(* Logix 5000 project; controller RN21_Architecture 1769-L16ER-BB1B rev 35.11; software revision 35.00; part 8 of 9 *)
(* tags used below, declared in another part *)
   ANM_C1Pause_Release : BOOL;
   ANM_C1StartReq : BOOL;
   ANM_C1StopReq_Auto : BOOL;
   ANM_C1StopReq_HMI : BOOL;
   ANM_C2Pause_Release : BOOL;
   ANM_C2StartReq : BOOL;
   ANM_C2StopReq_Auto : BOOL;
   ANM_C2StopReq_HMI : BOOL;
   ANM_C3Pause_Release : BOOL;
   ANM_C3StartReq : BOOL;
   ANM_C3StopReq_Auto : BOOL;
   ANM_C3StopReq_HMI : BOOL;
   ANM_C4Pause_Release : BOOL;
   ANM_C4StartReq : BOOL;
   ANM_C4StopReq_Auto : BOOL;
   ANM_C4StopReq_HMI : BOOL;
   ANM_C5Pause_Release : BOOL;
   ANM_C5StartReq : BOOL;
   ANM_C5StopReq_Auto : BOOL;
   ANM_C5StopReq_HMI : BOOL;
   ANM_CStopReq_Alarm : BOOL;
   ANM_CycleReset : BOOL;
   BIT_RESET_TMR : TIMER;
   EmgLoginDn : BOOL;
   EnableInactivity : DINT;
   FC_LB_Arch : AOI_LOGIN_Arch;
   FC_PDL_Arch : AOI_PDL_Arch;
   FC_PDL_DC : AOI_PDL_DataCapture[10];
   FCI_ALARM : BOOL;
   FCI_AlarmReset : BOOL;
   FCI_C1COMPLETED : BOOL;
   FCI_C2COMPLETED : BOOL;
   FCI_C2PAUSE_RELEASE : BOOL;
   FCI_C2START : BOOL;
   FCI_C2STOP : BOOL;
   FCI_C3COMPLETED : BOOL;
   FCI_C3PAUSE_RELEASE : BOOL;
   FCI_C3START : BOOL;
   FCI_C3STOP : BOOL;
   FCI_C4COMPLETED : BOOL;
   FCI_C4PAUSE_RELEASE : BOOL;
   FCI_C4START : BOOL;
   FCI_C4STOP : BOOL;
   FCI_C5COMPLETED : BOOL;
   FCI_C5PAUSE_RELEASE : BOOL;
   FCI_C5STARTED : BOOL;
   FCI_C5STOP : BOOL;
   FCI_LBDataLogTrig : BOOL;
   FCI_PDLDataLogTrig : BOOL;
   FCI_PrintInterval : INT;
   FCI_PROCESSRESET : BOOL;
   FCO_C1CMPLTSTSMOVTRIG : BOOL;
   FCO_C1PAUSED : BOOL;
   FCO_C1PAUSEDSTSMOVTRIG : BOOL;
   FCO_C1RELEASEDSTSMOVTRIG : BOOL;
   FCO_C1RUNNINGSTSMOVTRIG : BOOL;
   FCO_C1STOPEDALMSTSMOVTRIG : BOOL;
   FCO_C1STOPEDSTSMOVTRIG : BOOL;
   FCO_C2CMPLTSTSMOVTRIG : BOOL;
   FCO_C2PAUSED : BOOL;
   FCO_C2PAUSEDSTSMOVTRIG : BOOL;
   FCO_C2RELEASEDSTSMOVTRIG : BOOL;
   FCO_C2RUNNINGSTSMOVTRIG : BOOL;
   FCO_C2STARTED : BOOL;
   FCO_C2STOPEDALMSTSMOVTRIG : BOOL;
   FCO_C2STOPEDSTSMOVTRIG : BOOL;
   FCO_C3CMPLTSTSMOVTRIG : BOOL;
   FCO_C3PAUSED : BOOL;
   FCO_C3PAUSEDSTSMOVTRIG : BOOL;
   FCO_C3RELEASEDSTSMOVTRIG : BOOL;
   FCO_C3RUNNINGSTSMOVTRIG : BOOL;
   FCO_C3STARTED : BOOL;
   FCO_C3STOPEDALMSTSMOVTRIG : BOOL;
   FCO_C3STOPEDSTSMOVTRIG : BOOL;
   FCO_C4CMPLTSTSMOVTRIG : BOOL;
   FCO_C4PAUSED : BOOL;
   FCO_C4PAUSEDSTSMOVTRIG : BOOL;
   FCO_C4RELEASEDSTSMOVTRIG : BOOL;
   FCO_C4RUNNINGSTSMOVTRIG : BOOL;
   FCO_C4STARTED : BOOL;
   FCO_C4STOPEDALMSTSMOVTRIG : BOOL;
   FCO_C4STOPEDSTSMOVTRIG : BOOL;
   FCO_C5CMPLTSTSMOVTRIG : BOOL;
   FCO_C5PAUSED : BOOL;
   FCO_C5PAUSEDSTSMOVTRIG : BOOL;
   FCO_C5RELEASEDSTSMOVTRIG : BOOL;
   FCO_C5RUNNINGSTSMOVTRIG : BOOL;
   FCO_C5STARTED : BOOL;
   FCO_C5STOPEDALARMSTSMOVTRIG : BOOL;
   FCO_C5STOPEDSTSMOVTRIG : BOOL;
   INTERNAL_RN21_HB_PLC2ServerCommFailed : BOOL;
   InvalidBit : BOOL;
   LBSrc : UDT_Login;
   LBSrc_UniqueNum : DINT;
   Lockout_Visb : BOOL;
   PDL_Para1 : REAL;
   PDL_Para2 : REAL;
   PDL_Para3 : REAL;
   PDL_Para4 : REAL;
   PDLSrc : UDT_Process;
   PDLSrc_PDL_UID : DINT;
   PLC_RTC : DINT[7];
   PrintIntervalReq : BOOL;
   RN21_AutoLogedOut : BOOL;
   RN21_DC_Active : BOOL;
   RN21_DC_Enable : BOOL;
   RN21_LBONS : DINT[2];
   RN21_LBStatus : INT;   // Login Block Status
   RN21_LBStatus1 : DINT;
   RN21_PDL_OSTBit : BOOL;
   RN21_PDL_OSTTempInt : DINT;   // One Second Trig
   RN21_PDLMAPONS : DINT;
   RN21_PDLParam : REAL[20];
   RN21_PDLStatus : DINT;
   RN21_PDLTrig : DINT;
   RN21_PrintInterval : DINT;
   RN21_RM_BITRESET : BOOL;
   RN21_RM_HMICheck : BOOL;
   RN21_RM_HMICODE : STRING;
   RN21_RM_HMILoad : BOOL;
   RN21_RM_LOADBIT : BOOL;
   RN21_RM_LOADBTNVISB : BOOL;
   RN21_RM_LOADDLY_TMRBIT : BOOL;
   RN21_RM_LOADDLYBIT : BOOL;
   RN21_RM_LOADSTATUS : DINT;
   RN21_RM_LOADVISB : BOOL;
   RN21_RM_ONS : BOOL[64];
   RN21_RM_STATUS_VISB : BOOL;
   RN21_UM_Empty : STRING;   // Whenever Logout Will happen moving the Empty
   RN21_UM_HMIPSWD_Visb : BOOL;
   RN21_UM_UserLogout : BOOL;
   RN21_UMLogoutTag : INT;
   RN21_UserLoginDN : BOOL;
   teset : BOOL;
   TestProcessTag : REAL[8];
   TMR_AutoLogoutRstDly : TIMER;
   TMR_LOAD_DLY : TIMER;
   TMR_ONE_SECBIT_RST : TIMER;
   TMR_SvrConfrm_BIT : TIMER;
   UM_LogGenDelay : TIMER;
   EmergencyLoginActivated_Bit : BOOL;
   FCI_C1PAUSE_RELEASE : BOOL;
   FCI_C1START : BOOL;
   FCI_C1STOP : BOOL;
   FCO_C1STARTED : BOOL;
   LBSer : UDT_Login;
   LOGIN_TriggerId : BOOL;
   LOGIN_UniqueNum : DINT;
   PDL_Trigger : BOOL;
   PDL_UID : DINT;
   PDLSer : UDT_Process;
   RM_RecipeAck : DINT;
   RM_RecipeCode : STRING;
   RN21_PDLMainONS : BOOL;
   UM_Confirmation_Bit : BOOL;
   UM_lockoutDurationLeft : DINT;
   UM_Status : DINT;
   UM_UID : STRING;
(* MainProgram, continued *)

ROUTINE RN21_LB_Main   (* ladder *)
// User Management Architecture
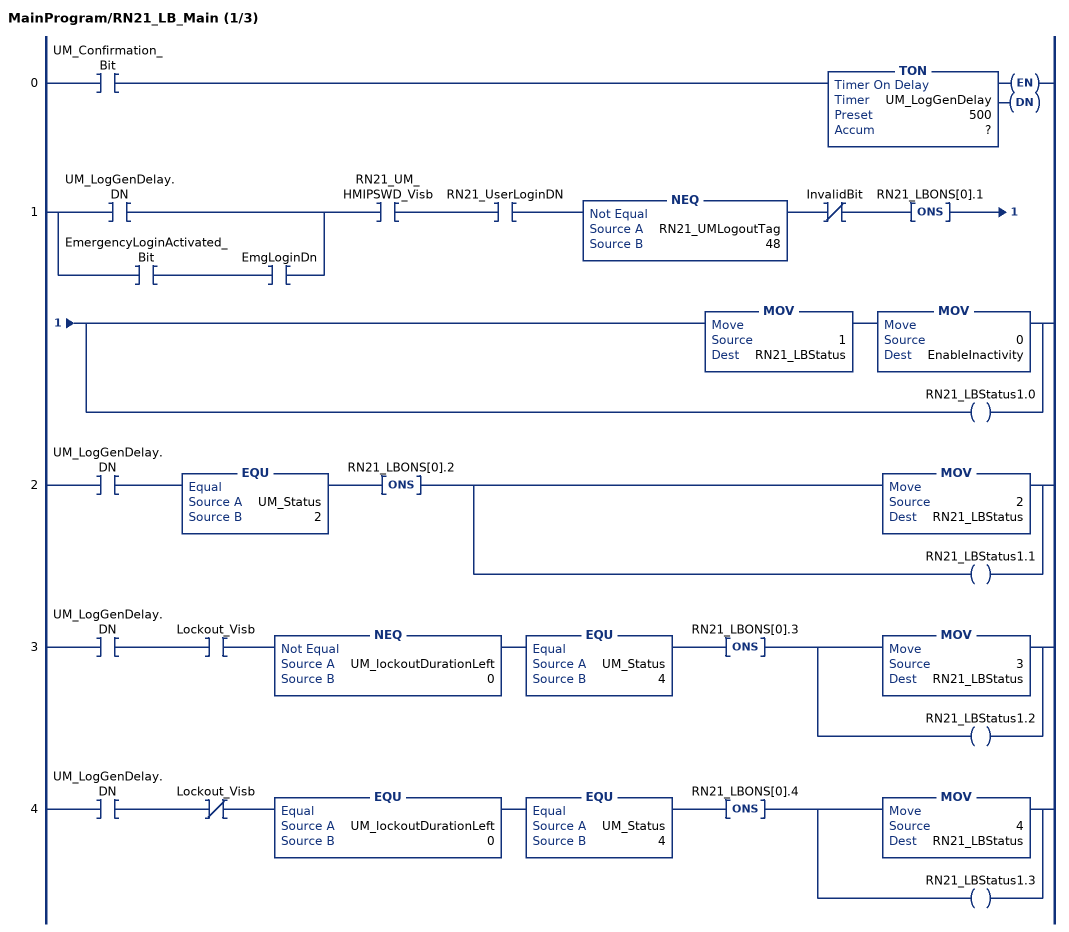
   0: XIC(UM_Confirmation_Bit)TON(UM_LogGenDelay,?,?);
   1: [XIC(UM_LogGenDelay.DN) ,XIC(EmergencyLoginActivated_Bit) XIC(EmgLoginDn) ]XIC(RN21_UM_HMIPSWD_Visb)XIC(RN21_UserLoginDN)NEQ(RN21_UMLogoutTag,48)XIO(InvalidBit)ONS(RN21_LBONS[0].1)[MOV(1,RN21_LBStatus) MOV(0,EnableInactivity) ,OTE(RN21_LBStatus1.0) ];
   2: XIC(UM_LogGenDelay.DN)EQU(UM_Status,2)ONS(RN21_LBONS[0].2)[MOV(2,RN21_LBStatus) ,OTE(RN21_LBStatus1.1) ];
   3: XIC(UM_LogGenDelay.DN)XIC(Lockout_Visb)NEQ(UM_lockoutDurationLeft,0)EQU(UM_Status,4)ONS(RN21_LBONS[0].3)[MOV(3,RN21_LBStatus) ,OTE(RN21_LBStatus1.2) ];
   4: XIC(UM_LogGenDelay.DN)XIO(Lockout_Visb)EQU(UM_lockoutDurationLeft,0)EQU(UM_Status,4)ONS(RN21_LBONS[0].4)[MOV(4,RN21_LBStatus) ,OTE(RN21_LBStatus1.3) ];
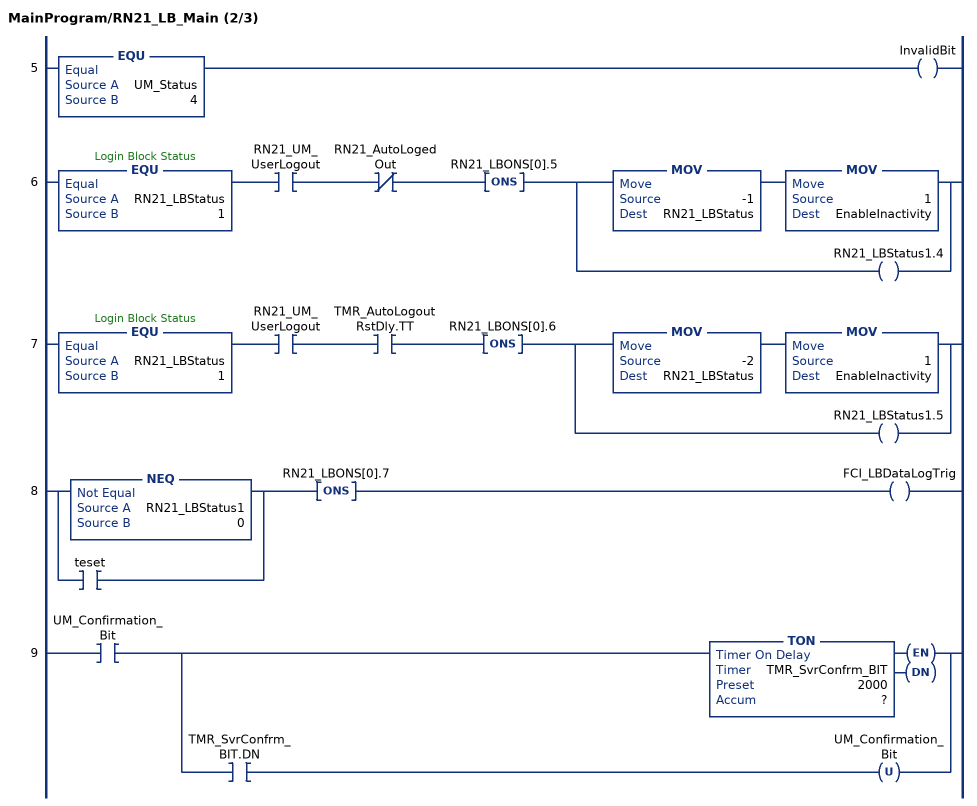
   5: EQU(UM_Status,4)OTE(InvalidBit);
   6: EQU(RN21_LBStatus,1)XIC(RN21_UM_UserLogout)XIO(RN21_AutoLogedOut)ONS(RN21_LBONS[0].5)[MOV(-1,RN21_LBStatus) MOV(1,EnableInactivity) ,OTE(RN21_LBStatus1.4) ];
   7: EQU(RN21_LBStatus,1)XIC(RN21_UM_UserLogout)XIC(TMR_AutoLogoutRstDly.TT)ONS(RN21_LBONS[0].6)[MOV(-2,RN21_LBStatus) MOV(1,EnableInactivity) ,OTE(RN21_LBStatus1.5) ];
   8: [NEQ(RN21_LBStatus1,0) ,XIC(teset) ]ONS(RN21_LBONS[0].7)OTE(FCI_LBDataLogTrig);
   9: XIC(UM_Confirmation_Bit)[TON(TMR_SvrConfrm_BIT,?,?) ,XIC(TMR_SvrConfrm_BIT.DN) OTU(UM_Confirmation_Bit) ];
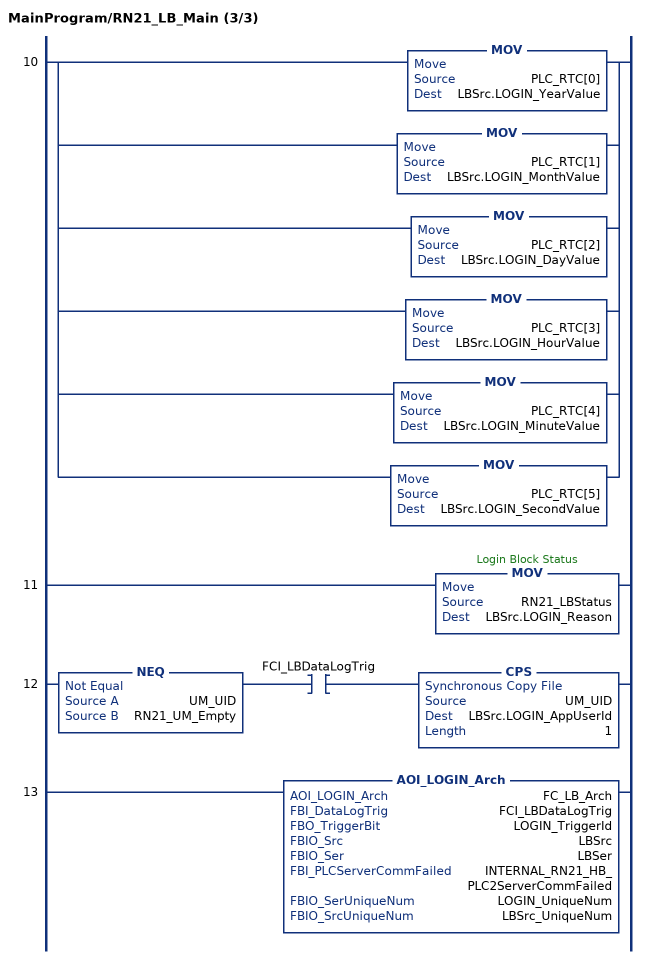
   10: [MOV(PLC_RTC[0],LBSrc.LOGIN_YearValue) ,MOV(PLC_RTC[1],LBSrc.LOGIN_MonthValue) ,MOV(PLC_RTC[2],LBSrc.LOGIN_DayValue) ,MOV(PLC_RTC[3],LBSrc.LOGIN_HourValue) ,MOV(PLC_RTC[4],LBSrc.LOGIN_MinuteValue) ,MOV(PLC_RTC[5],LBSrc.LOGIN_SecondValue) ];
   11: MOV(RN21_LBStatus,LBSrc.LOGIN_Reason);
   12: NEQ(UM_UID,RN21_UM_Empty)XIC(FCI_LBDataLogTrig)CPS(UM_UID,LBSrc.LOGIN_AppUserId,1);
   13: AOI_LOGIN_Arch(FC_LB_Arch,FCI_LBDataLogTrig,LOGIN_TriggerId,LBSrc,LBSer,INTERNAL_RN21_HB_PLC2ServerCommFailed,LOGIN_UniqueNum,LBSrc_UniqueNum);
END_ROUTINE

ROUTINE RN21_PDL_Main   (* ladder *)
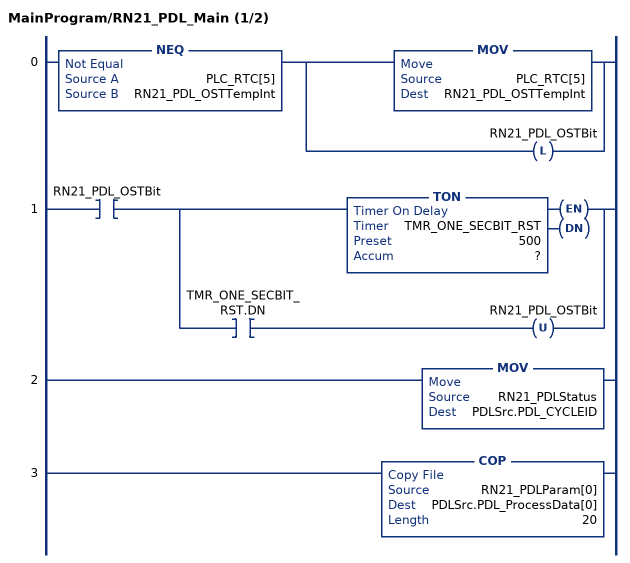
   0: NEQ(PLC_RTC[5],RN21_PDL_OSTTempInt)[MOV(PLC_RTC[5],RN21_PDL_OSTTempInt) ,OTL(RN21_PDL_OSTBit) ];
   1: XIC(RN21_PDL_OSTBit)[TON(TMR_ONE_SECBIT_RST,?,?) ,XIC(TMR_ONE_SECBIT_RST.DN) OTU(RN21_PDL_OSTBit) ];
   2: MOV(RN21_PDLStatus,PDLSrc.PDL_CYCLEID);
   3: COP(RN21_PDLParam[0],PDLSrc.PDL_ProcessData[0],20);
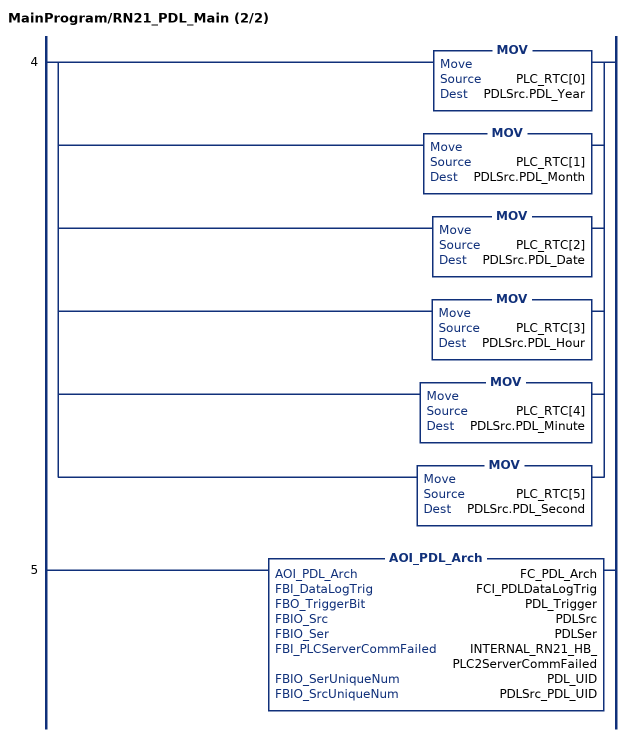
   4: [MOV(PLC_RTC[0],PDLSrc.PDL_Year) ,MOV(PLC_RTC[1],PDLSrc.PDL_Month) ,MOV(PLC_RTC[2],PDLSrc.PDL_Date) ,MOV(PLC_RTC[3],PDLSrc.PDL_Hour) ,MOV(PLC_RTC[4],PDLSrc.PDL_Minute) ,MOV(PLC_RTC[5],PDLSrc.PDL_Second) ];
   5: AOI_PDL_Arch(FC_PDL_Arch,FCI_PDLDataLogTrig,PDL_Trigger,PDLSrc,PDLSer,INTERNAL_RN21_HB_PLC2ServerCommFailed,PDL_UID,PDLSrc_PDL_UID);
END_ROUTINE

ROUTINE RN21_PDL_Map   (* ladder *)
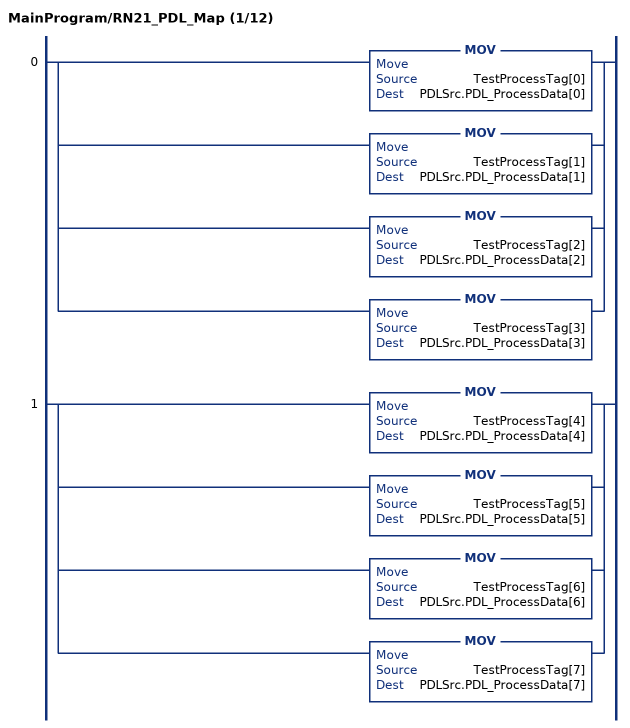
   0: [MOV(TestProcessTag[0],PDLSrc.PDL_ProcessData[0]) ,MOV(TestProcessTag[1],PDLSrc.PDL_ProcessData[1]) ,MOV(TestProcessTag[2],PDLSrc.PDL_ProcessData[2]) ,MOV(TestProcessTag[3],PDLSrc.PDL_ProcessData[3]) ];
   1: [MOV(TestProcessTag[4],PDLSrc.PDL_ProcessData[4]) ,MOV(TestProcessTag[5],PDLSrc.PDL_ProcessData[5]) ,MOV(TestProcessTag[6],PDLSrc.PDL_ProcessData[6]) ,MOV(TestProcessTag[7],PDLSrc.PDL_ProcessData[7]) ];
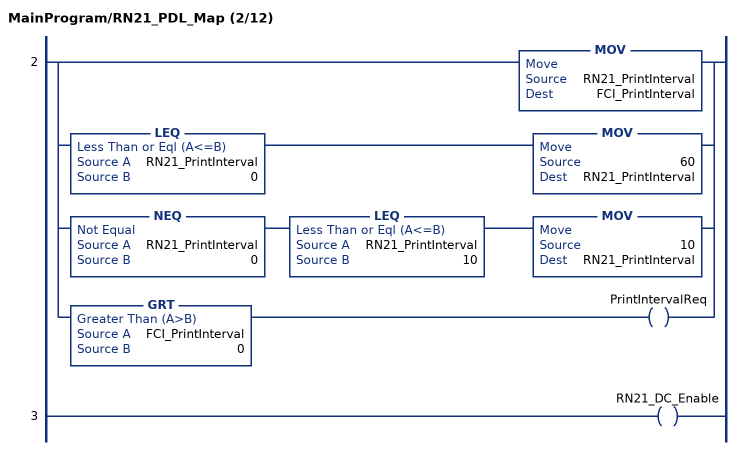
   2: [MOV(RN21_PrintInterval,FCI_PrintInterval) ,LEQ(RN21_PrintInterval,0) MOV(60,RN21_PrintInterval) ,NEQ(RN21_PrintInterval,0) LEQ(RN21_PrintInterval,10) MOV(10,RN21_PrintInterval) ,GRT(FCI_PrintInterval,0) OTE(PrintIntervalReq) ];
   3: OTE(RN21_DC_Enable);
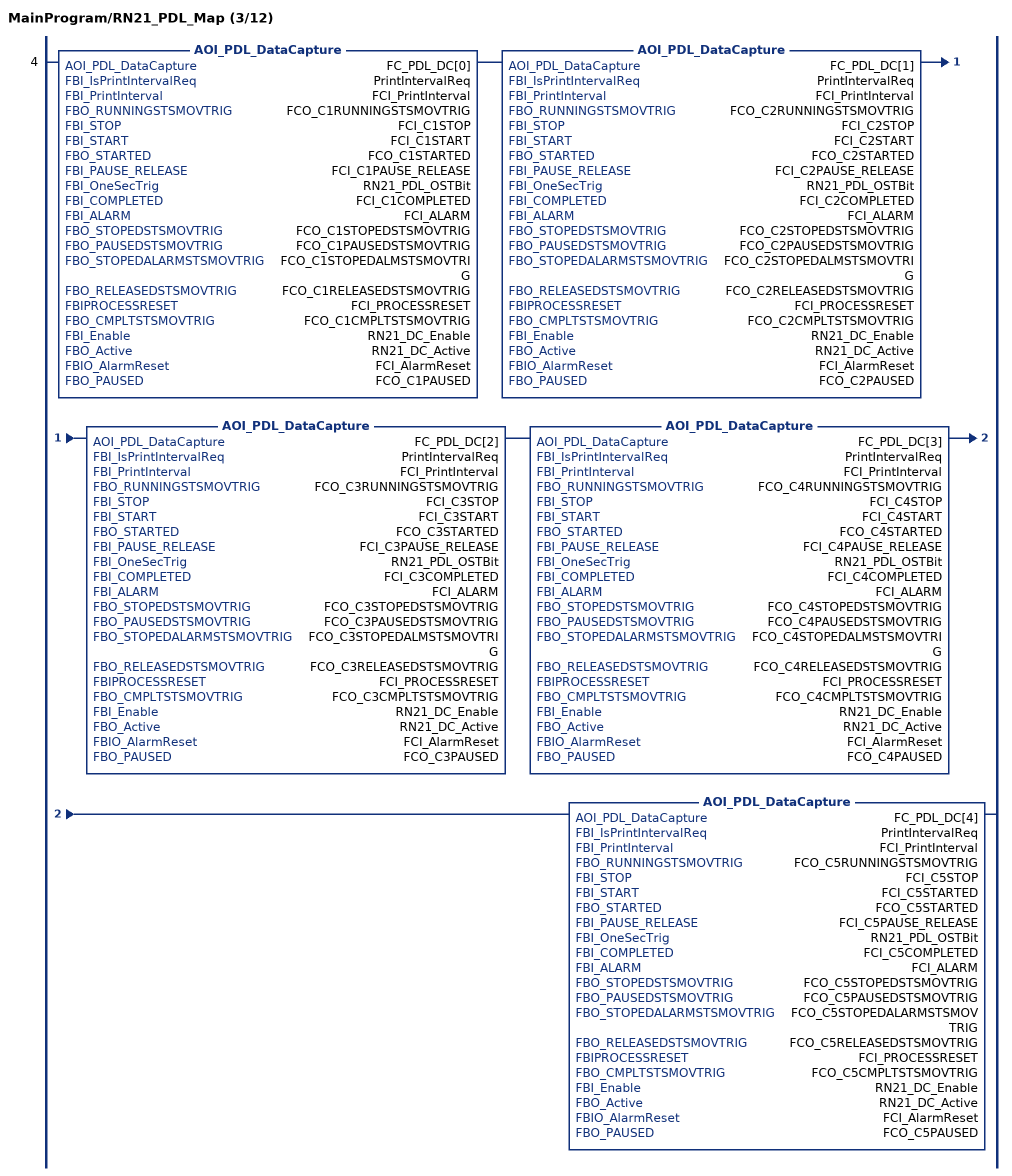
   4: AOI_PDL_DataCapture(FC_PDL_DC[0],PrintIntervalReq,FCI_PrintInterval,FCO_C1RUNNINGSTSMOVTRIG,FCI_C1STOP,FCI_C1START,FCO_C1STARTED,FCI_C1PAUSE_RELEASE,RN21_PDL_OSTBit,FCI_C1COMPLETED,FCI_ALARM,FCO_C1STOPEDSTSMOVTRIG,FCO_C1PAUSEDSTSMOVTRIG,FCO_C1STOPEDALMSTSMOVTRIG,FCO_C1RELEASEDSTSMOVTRIG,FCI_PROCESSRESET,FCO_C1CMPLTSTSMOVTRIG,RN21_DC_Enable,RN21_DC_Active,FCI_AlarmReset,FCO_C1PAUSED)AOI_PDL_DataCapture(FC_PDL_DC[1],PrintIntervalReq,FCI_PrintInterval,FCO_C2RUNNINGSTSMOVTRIG,FCI_C2STOP,FCI_C2START,FCO_C2STARTED,FCI_C2PAUSE_RELEASE,RN21_PDL_OSTBit,FCI_C2COMPLETED,FCI_ALARM,FCO_C2STOPEDSTSMOVTRIG,FCO_C2PAUSEDSTSMOVTRIG,FCO_C2STOPEDALMSTSMOVTRIG,FCO_C2RELEASEDSTSMOVTRIG,FCI_PROCESSRESET,FCO_C2CMPLTSTSMOVTRIG,RN21_DC_Enable,RN21_DC_Active,FCI_AlarmReset,FCO_C2PAUSED)AOI_PDL_DataCapture(FC_PDL_DC[2],PrintIntervalReq,FCI_PrintInterval,FCO_C3RUNNINGSTSMOVTRIG,FCI_C3STOP,FCI_C3START,FCO_C3STARTED,FCI_C3PAUSE_RELEASE,RN21_PDL_OSTBit,FCI_C3COMPLETED,FCI_ALARM,FCO_C3STOPEDSTSMOVTRIG,FCO_C3PAUSEDSTSMOVTRIG,FCO_C3STOPEDALMSTSMOVTRIG,FCO_C3RELEASEDSTSMOVTRIG,FCI_PROCESSRESET,FCO_C3CMPLTSTSMOVTRIG,RN21_DC_Enable,RN21_DC_Active,FCI_AlarmReset,FCO_C3PAUSED)AOI_PDL_DataCapture(FC_PDL_DC[3],PrintIntervalReq,FCI_PrintInterval,FCO_C4RUNNINGSTSMOVTRIG,FCI_C4STOP,FCI_C4START,FCO_C4STARTED,FCI_C4PAUSE_RELEASE,RN21_PDL_OSTBit,FCI_C4COMPLETED,FCI_ALARM,FCO_C4STOPEDSTSMOVTRIG,FCO_C4PAUSEDSTSMOVTRIG,FCO_C4STOPEDALMSTSMOVTRIG,FCO_C4RELEASEDSTSMOVTRIG,FCI_PROCESSRESET,FCO_C4CMPLTSTSMOVTRIG,RN21_DC_Enable,RN21_DC_Active,FCI_AlarmReset,FCO_C4PAUSED)AOI_PDL_DataCapture(FC_PDL_DC[4],PrintIntervalReq,FCI_PrintInterval,FCO_C5RUNNINGSTSMOVTRIG,FCI_C5STOP,FCI_C5STARTED,FCO_C5STARTED,FCI_C5PAUSE_RELEASE,RN21_PDL_OSTBit,FCI_C5COMPLETED,FCI_ALARM,FCO_C5STOPEDSTSMOVTRIG,FCO_C5PAUSEDSTSMOVTRIG,FCO_C5STOPEDALARMSTSMOVTRIG,FCO_C5RELEASEDSTSMOVTRIG,FCI_PROCESSRESET,FCO_C5CMPLTSTSMOVTRIG,RN21_DC_Enable,RN21_DC_Active,FCI_AlarmReset,FCO_C5PAUSED);
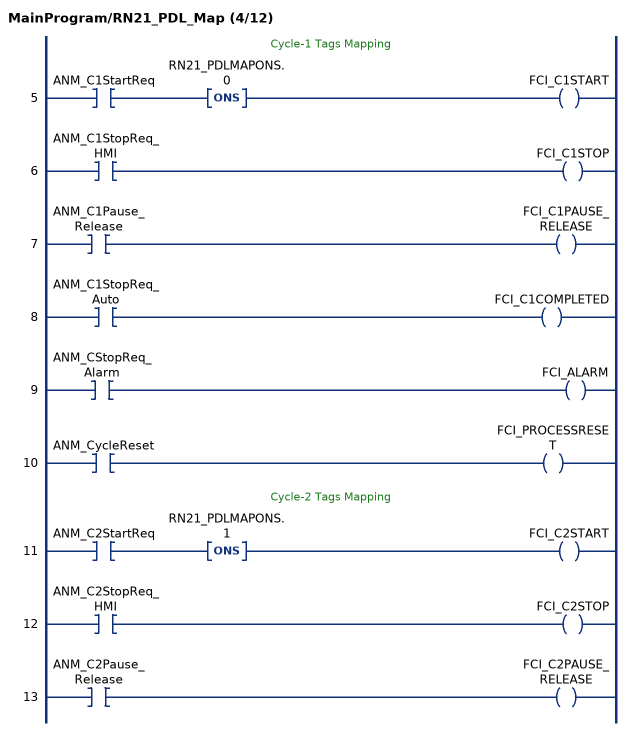
   // Cycle-1 Tags Mapping
   5: XIC(ANM_C1StartReq)ONS(RN21_PDLMAPONS.0)OTE(FCI_C1START);
   6: XIC(ANM_C1StopReq_HMI)OTE(FCI_C1STOP);
   7: XIC(ANM_C1Pause_Release)OTE(FCI_C1PAUSE_RELEASE);
   8: XIC(ANM_C1StopReq_Auto)OTE(FCI_C1COMPLETED);
   9: XIC(ANM_CStopReq_Alarm)OTE(FCI_ALARM);
   10: XIC(ANM_CycleReset)OTE(FCI_PROCESSRESET);
   // Cycle-2 Tags Mapping
   11: XIC(ANM_C2StartReq)ONS(RN21_PDLMAPONS.1)OTE(FCI_C2START);
   12: XIC(ANM_C2StopReq_HMI)OTE(FCI_C2STOP);
   13: XIC(ANM_C2Pause_Release)OTE(FCI_C2PAUSE_RELEASE);
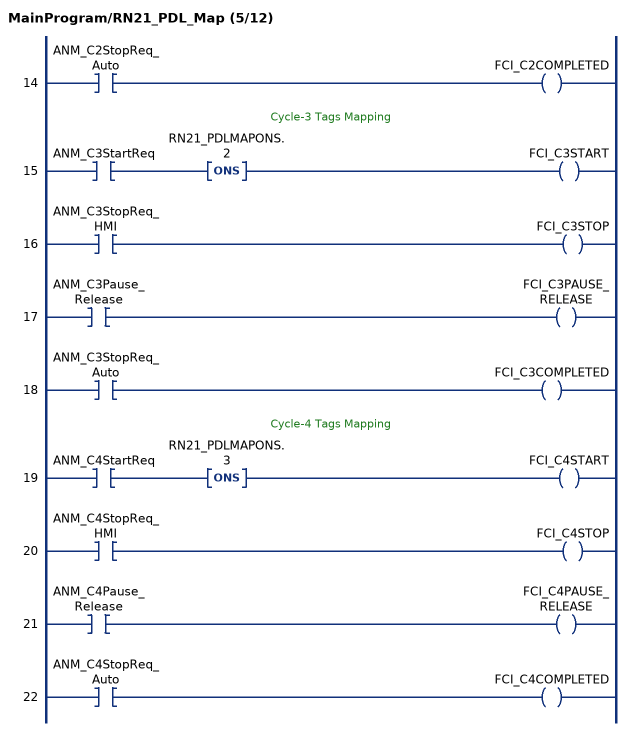
   14: XIC(ANM_C2StopReq_Auto)OTE(FCI_C2COMPLETED);
   // Cycle-3 Tags Mapping
   15: XIC(ANM_C3StartReq)ONS(RN21_PDLMAPONS.2)OTE(FCI_C3START);
   16: XIC(ANM_C3StopReq_HMI)OTE(FCI_C3STOP);
   17: XIC(ANM_C3Pause_Release)OTE(FCI_C3PAUSE_RELEASE);
   18: XIC(ANM_C3StopReq_Auto)OTE(FCI_C3COMPLETED);
   // Cycle-4 Tags Mapping
   19: XIC(ANM_C4StartReq)ONS(RN21_PDLMAPONS.3)OTE(FCI_C4START);
   20: XIC(ANM_C4StopReq_HMI)OTE(FCI_C4STOP);
   21: XIC(ANM_C4Pause_Release)OTE(FCI_C4PAUSE_RELEASE);
   22: XIC(ANM_C4StopReq_Auto)OTE(FCI_C4COMPLETED);
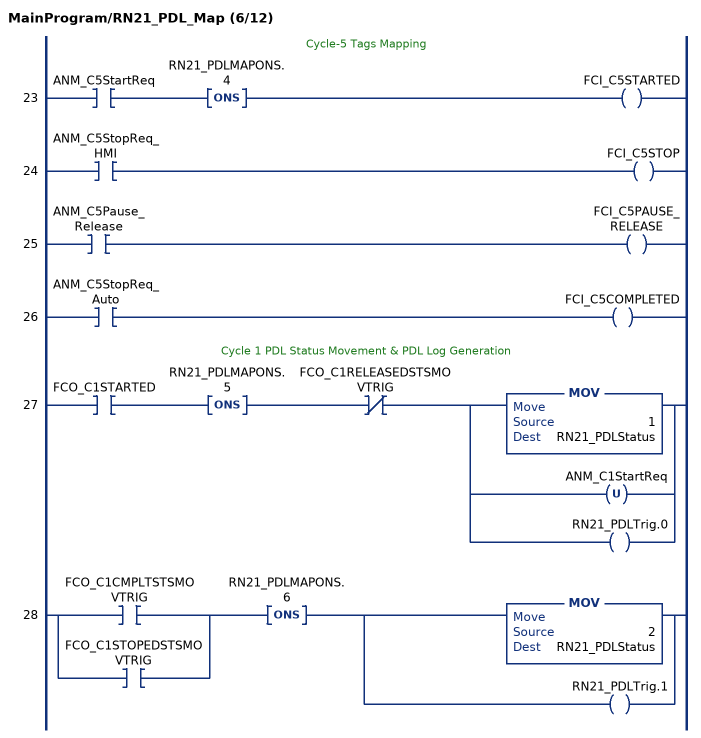
   // Cycle-5 Tags Mapping
   23: XIC(ANM_C5StartReq)ONS(RN21_PDLMAPONS.4)OTE(FCI_C5STARTED);
   24: XIC(ANM_C5StopReq_HMI)OTE(FCI_C5STOP);
   25: XIC(ANM_C5Pause_Release)OTE(FCI_C5PAUSE_RELEASE);
   26: XIC(ANM_C5StopReq_Auto)OTE(FCI_C5COMPLETED);
   // Cycle 1 PDL Status Movement & PDL Log Generation
   27: XIC(FCO_C1STARTED)ONS(RN21_PDLMAPONS.5)XIO(FCO_C1RELEASEDSTSMOVTRIG)[MOV(1,RN21_PDLStatus) ,OTU(ANM_C1StartReq) ,OTE(RN21_PDLTrig.0) ];
   28: [XIC(FCO_C1CMPLTSTSMOVTRIG) ,XIC(FCO_C1STOPEDSTSMOVTRIG) ]ONS(RN21_PDLMAPONS.6)[MOV(2,RN21_PDLStatus) ,OTE(RN21_PDLTrig.1) ];
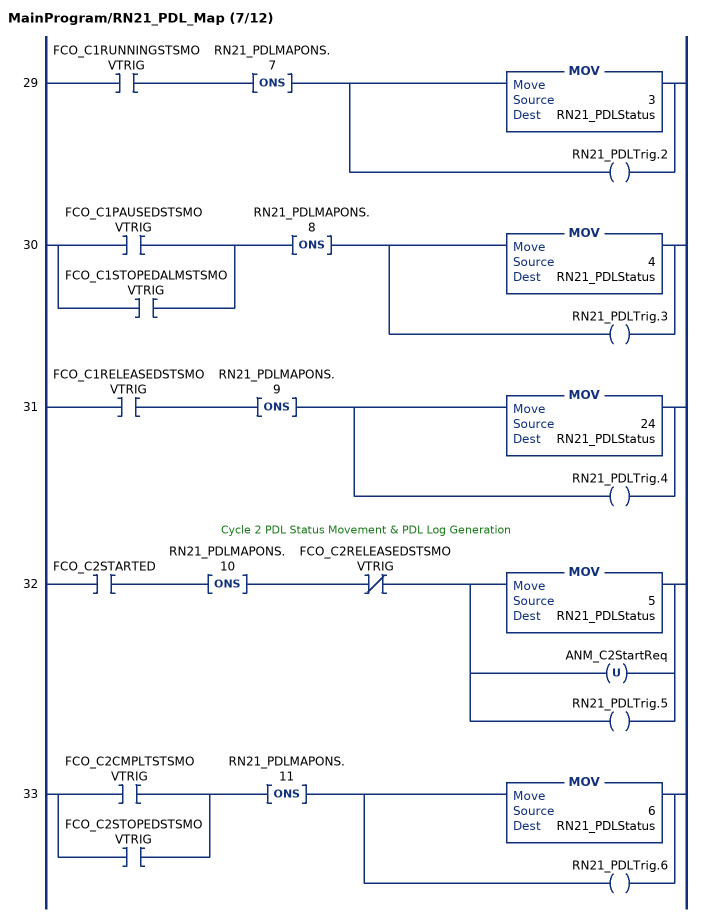
   29: XIC(FCO_C1RUNNINGSTSMOVTRIG)ONS(RN21_PDLMAPONS.7)[MOV(3,RN21_PDLStatus) ,OTE(RN21_PDLTrig.2) ];
   30: [XIC(FCO_C1PAUSEDSTSMOVTRIG) ,XIC(FCO_C1STOPEDALMSTSMOVTRIG) ]ONS(RN21_PDLMAPONS.8)[MOV(4,RN21_PDLStatus) ,OTE(RN21_PDLTrig.3) ];
   31: XIC(FCO_C1RELEASEDSTSMOVTRIG)ONS(RN21_PDLMAPONS.9)[MOV(24,RN21_PDLStatus) ,OTE(RN21_PDLTrig.4) ];
   // Cycle 2 PDL Status Movement & PDL Log Generation
   32: XIC(FCO_C2STARTED)ONS(RN21_PDLMAPONS.10)XIO(FCO_C2RELEASEDSTSMOVTRIG)[MOV(5,RN21_PDLStatus) ,OTU(ANM_C2StartReq) ,OTE(RN21_PDLTrig.5) ];
   33: [XIC(FCO_C2CMPLTSTSMOVTRIG) ,XIC(FCO_C2STOPEDSTSMOVTRIG) ]ONS(RN21_PDLMAPONS.11)[MOV(6,RN21_PDLStatus) ,OTE(RN21_PDLTrig.6) ];
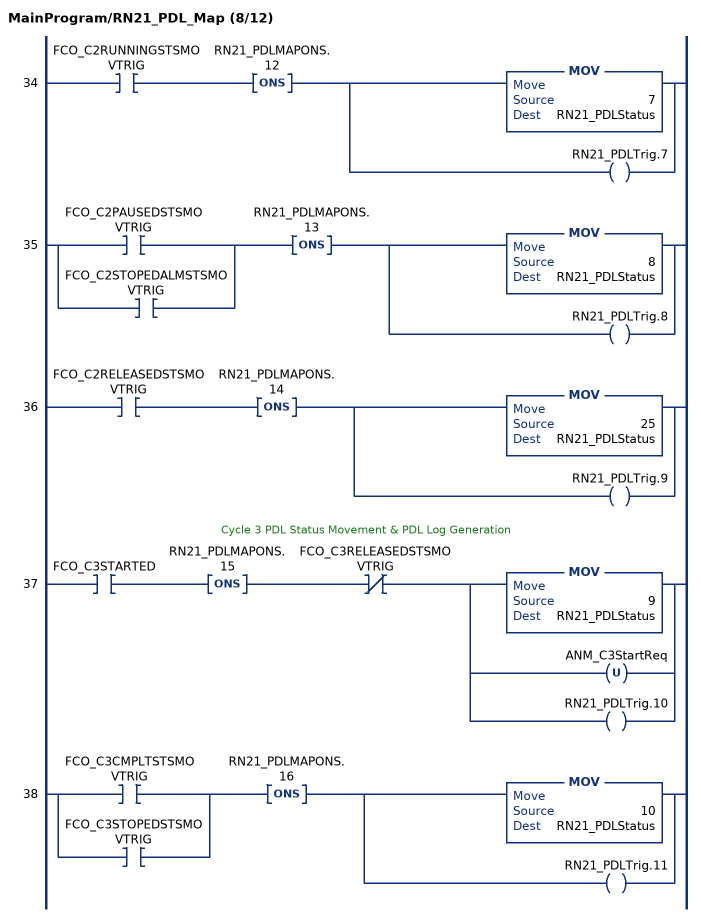
   34: XIC(FCO_C2RUNNINGSTSMOVTRIG)ONS(RN21_PDLMAPONS.12)[MOV(7,RN21_PDLStatus) ,OTE(RN21_PDLTrig.7) ];
   35: [XIC(FCO_C2PAUSEDSTSMOVTRIG) ,XIC(FCO_C2STOPEDALMSTSMOVTRIG) ]ONS(RN21_PDLMAPONS.13)[MOV(8,RN21_PDLStatus) ,OTE(RN21_PDLTrig.8) ];
   36: XIC(FCO_C2RELEASEDSTSMOVTRIG)ONS(RN21_PDLMAPONS.14)[MOV(25,RN21_PDLStatus) ,OTE(RN21_PDLTrig.9) ];
   // Cycle 3 PDL Status Movement & PDL Log Generation
   37: XIC(FCO_C3STARTED)ONS(RN21_PDLMAPONS.15)XIO(FCO_C3RELEASEDSTSMOVTRIG)[MOV(9,RN21_PDLStatus) ,OTU(ANM_C3StartReq) ,OTE(RN21_PDLTrig.10) ];
   38: [XIC(FCO_C3CMPLTSTSMOVTRIG) ,XIC(FCO_C3STOPEDSTSMOVTRIG) ]ONS(RN21_PDLMAPONS.16)[MOV(10,RN21_PDLStatus) ,OTE(RN21_PDLTrig.11) ];
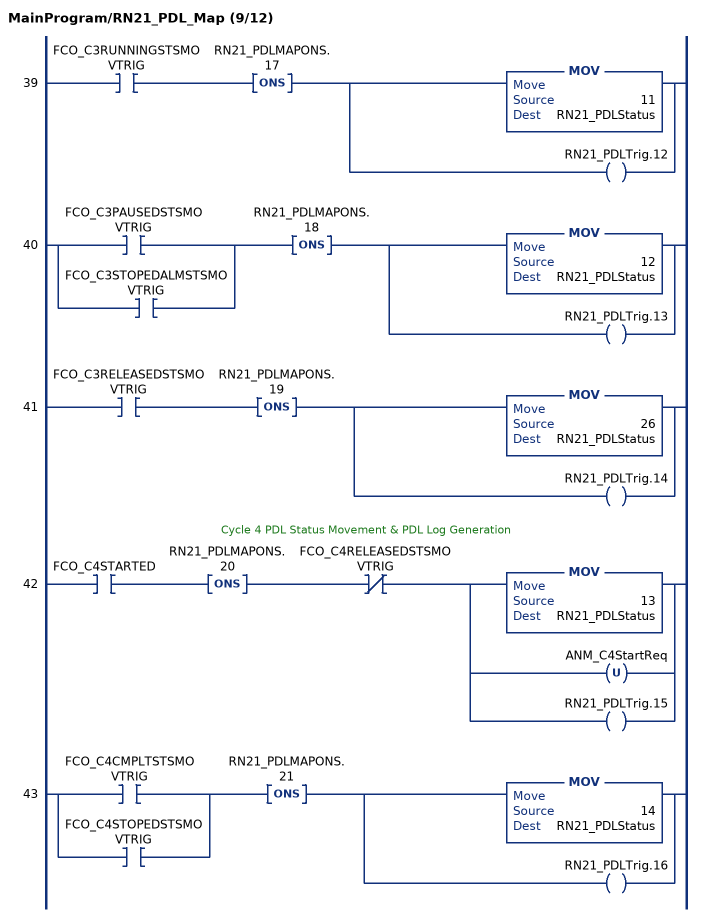
   39: XIC(FCO_C3RUNNINGSTSMOVTRIG)ONS(RN21_PDLMAPONS.17)[MOV(11,RN21_PDLStatus) ,OTE(RN21_PDLTrig.12) ];
   40: [XIC(FCO_C3PAUSEDSTSMOVTRIG) ,XIC(FCO_C3STOPEDALMSTSMOVTRIG) ]ONS(RN21_PDLMAPONS.18)[MOV(12,RN21_PDLStatus) ,OTE(RN21_PDLTrig.13) ];
   41: XIC(FCO_C3RELEASEDSTSMOVTRIG)ONS(RN21_PDLMAPONS.19)[MOV(26,RN21_PDLStatus) ,OTE(RN21_PDLTrig.14) ];
   // Cycle 4 PDL Status Movement & PDL Log Generation
   42: XIC(FCO_C4STARTED)ONS(RN21_PDLMAPONS.20)XIO(FCO_C4RELEASEDSTSMOVTRIG)[MOV(13,RN21_PDLStatus) ,OTU(ANM_C4StartReq) ,OTE(RN21_PDLTrig.15) ];
   43: [XIC(FCO_C4CMPLTSTSMOVTRIG) ,XIC(FCO_C4STOPEDSTSMOVTRIG) ]ONS(RN21_PDLMAPONS.21)[MOV(14,RN21_PDLStatus) ,OTE(RN21_PDLTrig.16) ];
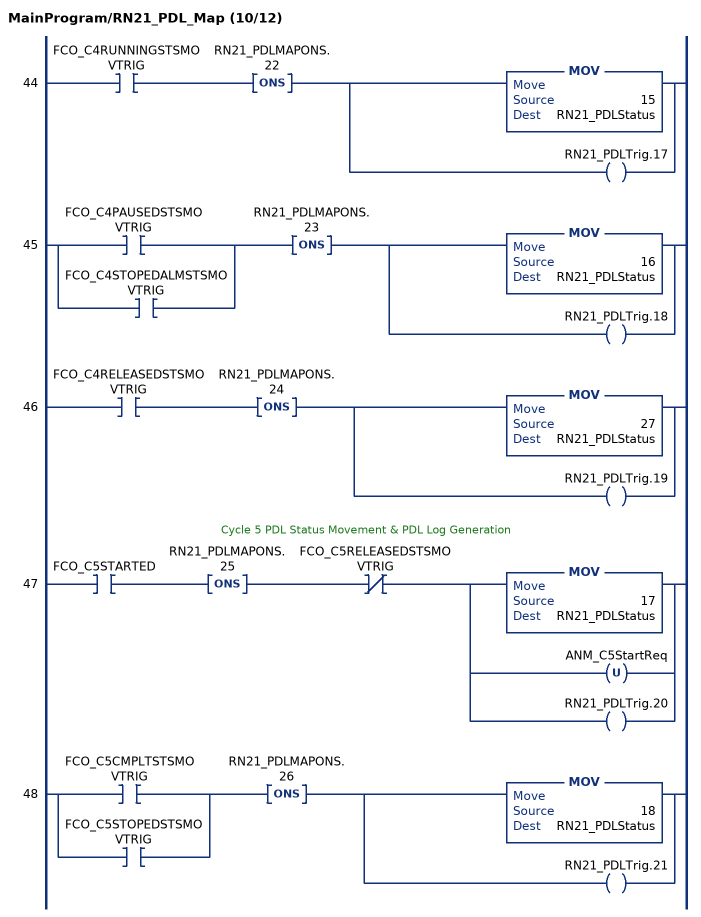
   44: XIC(FCO_C4RUNNINGSTSMOVTRIG)ONS(RN21_PDLMAPONS.22)[MOV(15,RN21_PDLStatus) ,OTE(RN21_PDLTrig.17) ];
   45: [XIC(FCO_C4PAUSEDSTSMOVTRIG) ,XIC(FCO_C4STOPEDALMSTSMOVTRIG) ]ONS(RN21_PDLMAPONS.23)[MOV(16,RN21_PDLStatus) ,OTE(RN21_PDLTrig.18) ];
   46: XIC(FCO_C4RELEASEDSTSMOVTRIG)ONS(RN21_PDLMAPONS.24)[MOV(27,RN21_PDLStatus) ,OTE(RN21_PDLTrig.19) ];
   // Cycle 5 PDL Status Movement & PDL Log Generation
   47: XIC(FCO_C5STARTED)ONS(RN21_PDLMAPONS.25)XIO(FCO_C5RELEASEDSTSMOVTRIG)[MOV(17,RN21_PDLStatus) ,OTU(ANM_C5StartReq) ,OTE(RN21_PDLTrig.20) ];
   48: [XIC(FCO_C5CMPLTSTSMOVTRIG) ,XIC(FCO_C5STOPEDSTSMOVTRIG) ]ONS(RN21_PDLMAPONS.26)[MOV(18,RN21_PDLStatus) ,OTE(RN21_PDLTrig.21) ];
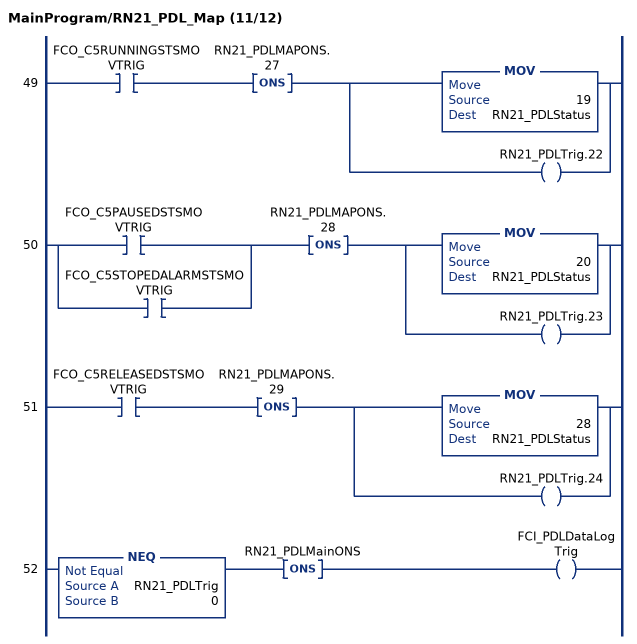
   49: XIC(FCO_C5RUNNINGSTSMOVTRIG)ONS(RN21_PDLMAPONS.27)[MOV(19,RN21_PDLStatus) ,OTE(RN21_PDLTrig.22) ];
   50: [XIC(FCO_C5PAUSEDSTSMOVTRIG) ,XIC(FCO_C5STOPEDALARMSTSMOVTRIG) ]ONS(RN21_PDLMAPONS.28)[MOV(20,RN21_PDLStatus) ,OTE(RN21_PDLTrig.23) ];
   51: XIC(FCO_C5RELEASEDSTSMOVTRIG)ONS(RN21_PDLMAPONS.29)[MOV(28,RN21_PDLStatus) ,OTE(RN21_PDLTrig.24) ];
   52: NEQ(RN21_PDLTrig,0)ONS(RN21_PDLMainONS)OTE(FCI_PDLDataLogTrig);
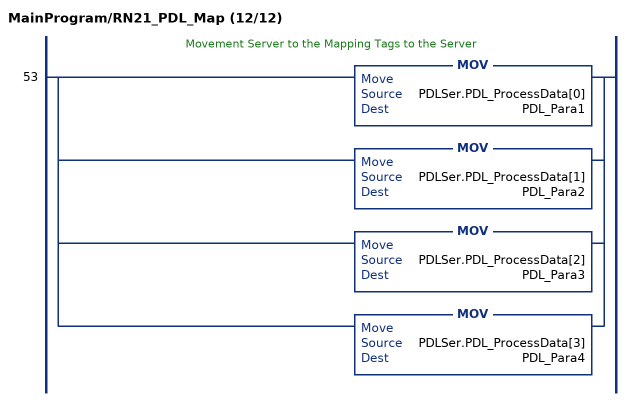
   // Movement Server to the Mapping Tags to the Server
   53: [MOV(PDLSer.PDL_ProcessData[0],PDL_Para1) ,MOV(PDLSer.PDL_ProcessData[1],PDL_Para2) ,MOV(PDLSer.PDL_ProcessData[2],PDL_Para3) ,MOV(PDLSer.PDL_ProcessData[3],PDL_Para4) ];
END_ROUTINE

ROUTINE RN21_RM_Main   (* ladder *)
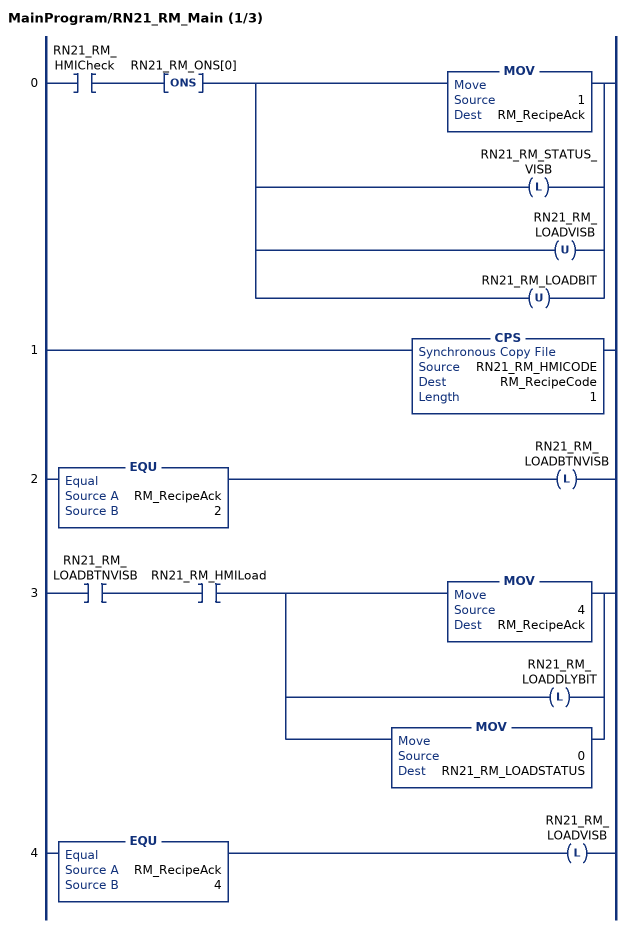
   0: XIC(RN21_RM_HMICheck)ONS(RN21_RM_ONS[0])[MOV(1,RM_RecipeAck) ,OTL(RN21_RM_STATUS_VISB) ,OTU(RN21_RM_LOADVISB) ,OTU(RN21_RM_LOADBIT) ];
   1: CPS(RN21_RM_HMICODE,RM_RecipeCode,1);
   2: EQU(RM_RecipeAck,2)OTL(RN21_RM_LOADBTNVISB);
   3: XIC(RN21_RM_LOADBTNVISB)XIC(RN21_RM_HMILoad)[MOV(4,RM_RecipeAck) ,OTL(RN21_RM_LOADDLYBIT) ,MOV(0,RN21_RM_LOADSTATUS) ];
   4: EQU(RM_RecipeAck,4)OTL(RN21_RM_LOADVISB);
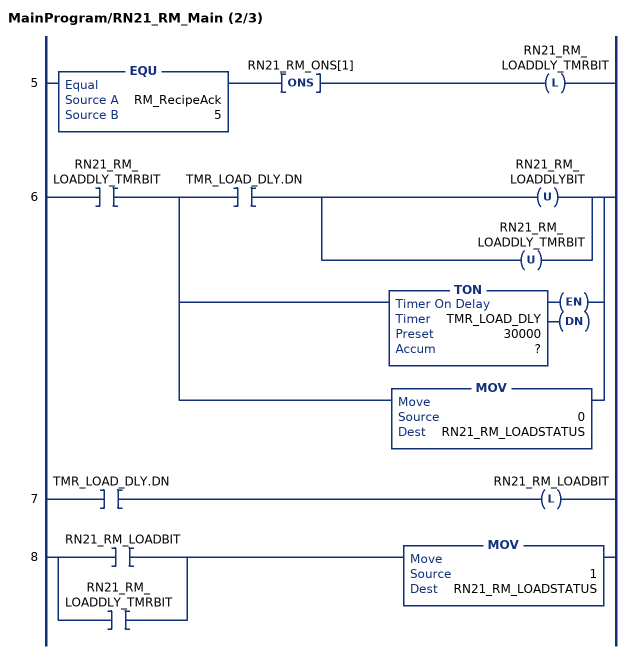
   5: EQU(RM_RecipeAck,5)ONS(RN21_RM_ONS[1])OTL(RN21_RM_LOADDLY_TMRBIT);
   6: XIC(RN21_RM_LOADDLY_TMRBIT)[XIC(TMR_LOAD_DLY.DN) [OTU(RN21_RM_LOADDLYBIT) ,OTU(RN21_RM_LOADDLY_TMRBIT) ] ,TON(TMR_LOAD_DLY,?,?) ,MOV(0,RN21_RM_LOADSTATUS) ];
   7: XIC(TMR_LOAD_DLY.DN)OTL(RN21_RM_LOADBIT);
   8: [XIC(RN21_RM_LOADBIT) ,XIC(RN21_RM_LOADDLY_TMRBIT) ]MOV(1,RN21_RM_LOADSTATUS);
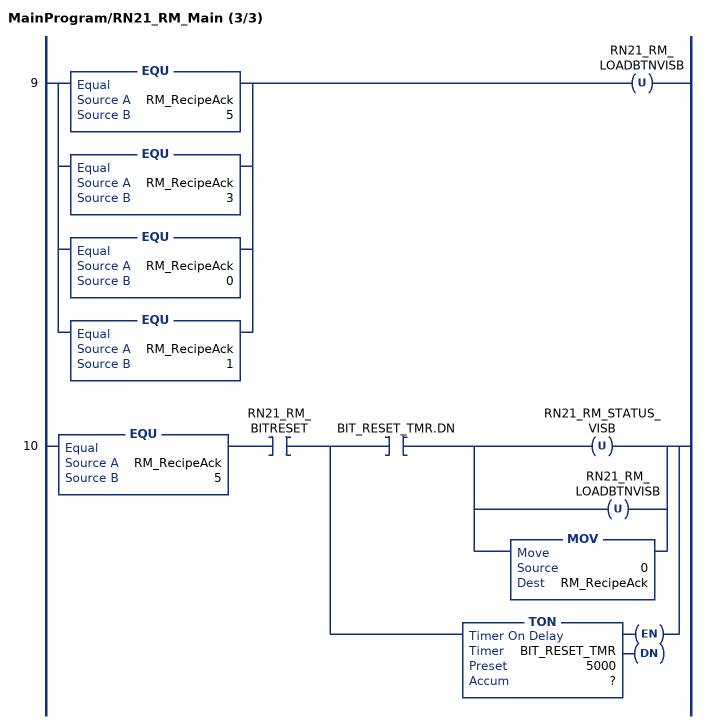
   9: [EQU(RM_RecipeAck,5) ,EQU(RM_RecipeAck,3) ,EQU(RM_RecipeAck,0) ,EQU(RM_RecipeAck,1) ]OTU(RN21_RM_LOADBTNVISB);
   10: EQU(RM_RecipeAck,5)XIC(RN21_RM_BITRESET)[XIC(BIT_RESET_TMR.DN) [[OTU(RN21_RM_STATUS_VISB) ,OTU(RN21_RM_LOADBTNVISB) ] ,MOV(0,RM_RecipeAck) ] ,TON(BIT_RESET_TMR,?,?) ];
END_ROUTINE
